{attribute 'qualified_only'}
VAR_GLOBAL
	bVR25On AT %Q* : BOOL := TRUE;
	bVR20On AT %Q* : BOOL := TRUE;
	
	iVR25Value AT %I* : INT;
	iVR20Value AT %I* : INT;
	
END_VAR

(* stored: Version 1.1.0.1, ProductVersion 3.1.4024.12
   GVL GVL: Id {11a8368a-ff2c-4c21-af16-feb83ec5ec04} *)
